Staubli VAL3: Rect3.dtx

public frame fReference = {x=1475.172, y=-187.34, z=-1030, rz=81.293, fatherId=world[0]}
public jointRx jPark = {j3=90, j5=90}
public jointRx jJoint = {j1=-21.01262, j2=66.00246, j3=79.8866, j5=34.11094, j6=162.86513}
public mdesc mNomSpeed = {blend=off}
public mdesc mSpeed[9]
  [0] = {tmax=75, rmax=100, leave=0.1, reach=0.1, blend=cartesian}
  [1] = {tmax=75, rmax=100, leave=0.1, reach=0.1, blend=cartesian}
  [2] = {tmax=75, rmax=100, leave=0.1, reach=0.1, blend=cartesian}
  [3] = {tmax=75, rmax=100, leave=0.1, reach=0.1, blend=cartesian}
  [4] = {tmax=75, rmax=100, leave=0.1, reach=0.1, blend=cartesian}
  [5] = {tmax=75, rmax=100, leave=0.1, reach=0.1, blend=cartesian}
  [6] = {tmax=75, rmax=100, leave=0.1, reach=0.1, blend=cartesian}
  [7] = {tmax=75, rmax=100, leave=0.1, reach=0.1, blend=cartesian}
  [8] = {tmax=75, rmax=100, leave=0.1, reach=0.1, blend=cartesian}
public num nTraj
num nTimeStop
num nTimeStart
num nMode
num nEtat
public pointRx pPoint[222]
  [0] = {x=-372, y=-44, z=100, rx=-180, rz=85.171, shoulder=lefty, elbow=epositive, wrist=wpositive, fatherId=fReference[0]}
  [1] = {x=-372, y=-44, rx=-180, rz=85.171, shoulder=lefty, elbow=epositive, wrist=wpositive, fatherId=fReference[0]}
  [2] = {x=-372, y=-44, rx=-180, rz=85.171, shoulder=lefty, elbow=epositive, wrist=wpositive, fatherId=fReference[0]}
  [3] = {x=-369.477, y=-73.864, rx=-180, rz=75.512, shoulder=lefty, elbow=epositive, wrist=wpositive, fatherId=fReference[0]}
  [4] = {x=-361.979, y=-102.881, rx=-180, rz=65.854, shoulder=lefty, elbow=epositive, wrist=wpositive, fatherId=fReference[0]}
  [5] = {x=-349.719, y=-130.229, rx=-180, rz=56.195, shoulder=lefty, elbow=epositive, wrist=wpositive, fatherId=fReference[0]}
  [6] = {x=-333.045, y=-155.133, rx=-180, rz=46.537, shoulder=lefty, elbow=epositive, wrist=wpositive, fatherId=fReference[0]}
  [7] = {x=-312.429, y=-176.886, rx=-180, rz=36.878, shoulder=lefty, elbow=epositive, wrist=wpositive, fatherId=fReference[0]}
  [8] = {x=-288.455, y=-194.872, rx=-180, rz=27.22, shoulder=lefty, elbow=epositive, wrist=wpositive, fatherId=fReference[0]}
  [9] = {x=-261.803, y=-208.58, rx=180, rz=17.561, shoulder=lefty, elbow=epositive, wrist=wpositive, fatherId=fReference[0]}
  [10] = {x=-233.23, y=-217.623, rx=-180, rz=7.903, shoulder=lefty, elbow=epositive, wrist=wpositive, fatherId=fReference[0]}
  [11] = {x=-203.544, y=-221.744, rx=180, rz=0.489, shoulder=lefty, elbow=epositive, wrist=wpositive, fatherId=fReference[0]}
  [12] = {x=-173.543, y=-222, rx=180, shoulder=lefty, elbow=epositive, wrist=wpositive, fatherId=fReference[0]}
  [13] = {x=-143.537, y=-222, rx=180, shoulder=lefty, elbow=epositive, wrist=wpositive, fatherId=fReference[0]}
  [14] = {x=-113.531, y=-222, rx=180, shoulder=lefty, elbow=epositive, wrist=wpositive, fatherId=fReference[0]}
  [15] = {x=-83.525, y=-222, rx=-180, shoulder=lefty, elbow=epositive, wrist=wpositive, fatherId=fReference[0]}
  [16] = {x=-53.519, y=-222, rx=180, shoulder=lefty, elbow=epositive, wrist=wpositive, fatherId=fReference[0]}
  [17] = {x=-23.513, y=-222, rx=180, shoulder=lefty, elbow=epositive, wrist=wpositive, fatherId=fReference[0]}
  [18] = {x=6.493, y=-222, rx=-180, shoulder=lefty, elbow=epositive, wrist=wpositive, fatherId=fReference[0]}
  [19] = {x=36.499, y=-222, rx=180, shoulder=lefty, elbow=epositive, wrist=wpositive, fatherId=fReference[0]}
  [20] = {x=66.504, y=-222, rx=180, shoulder=lefty, elbow=epositive, wrist=wpositive, fatherId=fReference[0]}
  [21] = {x=96.51, y=-222, rx=180, shoulder=lefty, elbow=epositive, wrist=wpositive, fatherId=fReference[0]}
  [22] = {x=126.516, y=-222, rx=180, shoulder=lefty, elbow=epositive, wrist=wpositive, fatherId=fReference[0]}
  [23] = {x=156.522, y=-222, rx=-180, shoulder=lefty, elbow=epositive, wrist=wpositive, fatherId=fReference[0]}
  [24] = {x=186.528, y=-222, rx=-180, rz=-2.723, shoulder=lefty, elbow=epositive, wrist=wpositive, fatherId=fReference[0]}
  [25] = {x=216.474, y=-220.576, rx=-180, rz=-12.083, shoulder=lefty, elbow=epositive, wrist=wpositive, fatherId=fReference[0]}
  [26] = {x=245.78, y=-214.302, rx=180, rz=-21.741, shoulder=lefty, elbow=epositive, wrist=wpositive, fatherId=fReference[0]}
  [27] = {x=273.619, y=-203.201, rx=-180, rz=-31.4, shoulder=lefty, elbow=epositive, wrist=wpositive, fatherId=fReference[0]}
  [28] = {x=299.2, y=-187.586, rx=180, rz=-41.058, shoulder=lefty, elbow=epositive, wrist=wpositive, fatherId=fReference[0]}
  [29] = {x=321.799, y=-167.901, rx=180, rz=-50.717, shoulder=lefty, elbow=epositive, wrist=wpositive, fatherId=fReference[0]}
  [30] = {x=340.775, y=-144.703, rx=180, rz=-60.375, shoulder=lefty, elbow=epositive, wrist=wpositive, fatherId=fReference[0]}
  [31] = {x=355.59, y=-118.65, rx=-180, rz=-70.034, shoulder=lefty, elbow=epositive, wrist=wpositive, fatherId=fReference[0]}
  [32] = {x=365.824, y=-90.481, rx=180, rz=-79.692, shoulder=lefty, elbow=epositive, wrist=wpositive, fatherId=fReference[0]}
  [33] = {x=371.187, y=-60.995, rx=180, rz=-88.446, shoulder=lefty, elbow=epositive, wrist=wpositive, fatherId=fReference[0]}
  [34] = {x=372, y=-31.015, rx=180, rz=-90, shoulder=lefty, elbow=epositive, wrist=wpositive, fatherId=fReference[0]}
  [35] = {x=372, y=-1.009, rx=180, rz=-90, shoulder=lefty, elbow=epositive, wrist=wpositive, fatherId=fReference[0]}
  [36] = {x=372, y=28.997, rx=-180, rz=-91.207, shoulder=lefty, elbow=epositive, wrist=wpositive, fatherId=fReference[0]}
  [37] = {x=371.368, y=58.985, rx=-180, rz=-99.658, shoulder=lefty, elbow=epositive, wrist=wpositive, fatherId=fReference[0]}
  [38] = {x=366.34, y=88.531, rx=-180, rz=-109.317, shoulder=lefty, elbow=epositive, wrist=wpositive, fatherId=fReference[0]}
  [39] = {x=356.426, y=116.814, rx=-180, rz=-118.975, shoulder=lefty, elbow=epositive, wrist=wpositive, fatherId=fReference[0]}
  [40] = {x=341.907, y=143.033, rx=-180, rz=-128.634, shoulder=lefty, elbow=epositive, wrist=wpositive, fatherId=fReference[0]}
  [41] = {x=323.195, y=166.444, rx=-180, rz=-138.292, shoulder=lefty, elbow=epositive, wrist=wpositive, fatherId=fReference[0]}
  [42] = {x=300.821, y=186.384, rx=180, rz=-147.951, shoulder=lefty, elbow=epositive, wrist=wpositive, fatherId=fReference[0]}
  [43] = {x=275.418, y=202.288, rx=180, rz=-157.609, shoulder=lefty, elbow=epositive, wrist=wpositive, fatherId=fReference[0]}
  [44] = {x=247.707, y=213.704, rx=-180, rz=-167.268, shoulder=lefty, elbow=epositive, wrist=wpositive, fatherId=fReference[0]}
  [45] = {x=218.474, y=220.309, rx=-180, rz=-176.767, shoulder=lefty, elbow=epositive, wrist=wpositive, fatherId=fReference[0]}
  [46] = {x=188.546, y=222, rx=-180, rz=180, shoulder=lefty, elbow=epositive, wrist=wpositive, fatherId=fReference[0]}
  [47] = {x=158.54, y=222, rx=-180, rz=180, shoulder=lefty, elbow=epositive, wrist=wpositive, fatherId=fReference[0]}
  [48] = {x=128.534, y=222, rx=180, rz=180, shoulder=lefty, elbow=epositive, wrist=wpositive, fatherId=fReference[0]}
  [49] = {x=98.528, y=222, rx=-180, rz=180, shoulder=lefty, elbow=epositive, wrist=wpositive, fatherId=fReference[0]}
  [50] = {x=68.522, y=222, rx=180, rz=180, shoulder=lefty, elbow=epositive, wrist=wpositive, fatherId=fReference[0]}
  [51] = {x=38.516, y=222, rx=-180, rz=180, shoulder=lefty, elbow=epositive, wrist=wpositive, fatherId=fReference[0]}
  [52] = {x=8.51, y=222, rx=-180, rz=180, shoulder=lefty, elbow=epositive, wrist=wpositive, fatherId=fReference[0]}
  [53] = {x=-21.496, y=222, rx=-180, rz=180, shoulder=lefty, elbow=epositive, wrist=wpositive, fatherId=fReference[0]}
  [54] = {x=-51.501, y=222, rx=-180, rz=180, shoulder=lefty, elbow=epositive, wrist=wpositive, fatherId=fReference[0]}
  [55] = {x=-81.507, y=222, rx=180, rz=180, shoulder=lefty, elbow=epositive, wrist=wpositive, fatherId=fReference[0]}
  [56] = {x=-111.513, y=222, rx=180, rz=-180, shoulder=lefty, elbow=epositive, wrist=wpositive, fatherId=fReference[0]}
  [57] = {x=-141.519, y=222, rx=180, rz=180, shoulder=lefty, elbow=epositive, wrist=wpositive, fatherId=fReference[0]}
  [58] = {x=-171.525, y=222, rx=-180, rz=179.696, shoulder=lefty, elbow=epositive, wrist=wpositive, fatherId=fReference[0]}
  [59] = {x=-201.529, y=221.841, rx=-180, rz=172.747, shoulder=lefty, elbow=epositive, wrist=wpositive, fatherId=fReference[0]}
  [60] = {x=-231.259, y=218.057, rx=-180, rz=163.088, shoulder=lefty, elbow=epositive, wrist=wpositive, fatherId=fReference[0]}
  [61] = {x=-259.934, y=209.338, rx=180, rz=153.43, shoulder=lefty, elbow=epositive, wrist=wpositive, fatherId=fReference[0]}
  [62] = {x=-286.739, y=195.933, rx=-180, rz=143.771, shoulder=lefty, elbow=epositive, wrist=wpositive, fatherId=fReference[0]}
  [63] = {x=-310.915, y=178.22, rx=180, rz=134.113, shoulder=lefty, elbow=epositive, wrist=wpositive, fatherId=fReference[0]}
  [64] = {x=-331.776, y=156.702, rx=180, rz=124.454, shoulder=lefty, elbow=epositive, wrist=wpositive, fatherId=fReference[0]}
  [65] = {x=-348.732, y=131.989, rx=180, rz=114.796, shoulder=lefty, elbow=epositive, wrist=wpositive, fatherId=fReference[0]}
  [66] = {x=-361.301, y=104.782, rx=180, rz=105.137, shoulder=lefty, elbow=epositive, wrist=wpositive, fatherId=fReference[0]}
  [67] = {x=-369.127, y=75.851, rx=180, rz=95.479, shoulder=lefty, elbow=epositive, wrist=wpositive, fatherId=fReference[0]}
  [68] = {x=-371.989, y=46.018, rx=180, rz=90.022, shoulder=lefty, elbow=epositive, wrist=wpositive, fatherId=fReference[0]}
  [69] = {x=-372, y=16.012, rx=-180, rz=90, shoulder=lefty, elbow=epositive, wrist=wpositive, fatherId=fReference[0]}
  [70] = {x=-372, y=-13.994, rx=-180, rz=90, shoulder=lefty, elbow=epositive, wrist=wpositive, fatherId=fReference[0]}
  [71] = {x=-372, y=-44, rx=-180, rz=90, shoulder=lefty, elbow=epositive, wrist=wpositive, fatherId=fReference[0]}
  [72] = {x=-372, y=-44, rx=-180, rz=90, shoulder=lefty, elbow=epositive, wrist=wpositive, fatherId=fReference[0]}
  [73] = {x=-372, y=-44, z=100, rx=-180, rz=90, shoulder=lefty, elbow=epositive, wrist=wpositive, fatherId=fReference[0]}
  [74] = {x=-372, y=-44, z=122, rx=-180, rz=90, shoulder=lefty, elbow=epositive, wrist=wpositive, fatherId=fReference[0]}
  [75] = {x=-372, y=-44, z=22, rx=-180, rz=90, shoulder=lefty, elbow=epositive, wrist=wpositive, fatherId=fReference[0]}
  [76] = {x=-372, y=-44, z=22, rx=-180, rz=90, shoulder=lefty, elbow=epositive, wrist=wpositive, fatherId=fReference[0]}
  [77] = {x=-372, y=-13.994, z=22, rx=-180, rz=90, shoulder=lefty, elbow=epositive, wrist=wpositive, fatherId=fReference[0]}
  [78] = {x=-372, y=16.012, z=22, rx=180, rz=90.022, shoulder=lefty, elbow=epositive, wrist=wpositive, fatherId=fReference[0]}
  [79] = {x=-371.989, y=46.018, z=22, rx=180, rz=95.479, shoulder=lefty, elbow=epositive, wrist=wpositive, fatherId=fReference[0]}
  [80] = {x=-369.127, y=75.851, z=22, rx=180, rz=105.137, shoulder=lefty, elbow=epositive, wrist=wpositive, fatherId=fReference[0]}
  [81] = {x=-361.301, y=104.782, z=22, rx=180, rz=114.796, shoulder=lefty, elbow=epositive, wrist=wpositive, fatherId=fReference[0]}
  [82] = {x=-348.732, y=131.989, z=22, rx=180, rz=124.454, shoulder=lefty, elbow=epositive, wrist=wpositive, fatherId=fReference[0]}
  [83] = {x=-331.776, y=156.702, z=22, rx=180, rz=134.113, shoulder=lefty, elbow=epositive, wrist=wpositive, fatherId=fReference[0]}
  [84] = {x=-310.915, y=178.22, z=22, rx=180, rz=143.771, shoulder=lefty, elbow=epositive, wrist=wpositive, fatherId=fReference[0]}
  [85] = {x=-286.739, y=195.933, z=22, rx=-180, rz=153.43, shoulder=lefty, elbow=epositive, wrist=wpositive, fatherId=fReference[0]}
  [86] = {x=-259.934, y=209.338, z=22, rx=-180, rz=163.088, shoulder=lefty, elbow=epositive, wrist=wpositive, fatherId=fReference[0]}
  [87] = {x=-231.259, y=218.057, z=22, rx=180, rz=172.747, shoulder=lefty, elbow=epositive, wrist=wpositive, fatherId=fReference[0]}
  [88] = {x=-201.529, y=221.841, z=22, rx=180, rz=179.696, shoulder=lefty, elbow=epositive, wrist=wpositive, fatherId=fReference[0]}
  [89] = {x=-171.525, y=222, z=22, rx=180, rz=180, shoulder=lefty, elbow=epositive, wrist=wpositive, fatherId=fReference[0]}
  [90] = {x=-141.519, y=222, z=22, rx=-180, rz=180, shoulder=lefty, elbow=epositive, wrist=wpositive, fatherId=fReference[0]}
  [91] = {x=-111.513, y=222, z=22, rx=180, rz=-180, shoulder=lefty, elbow=epositive, wrist=wpositive, fatherId=fReference[0]}
  [92] = {x=-81.507, y=222, z=22, rx=180, rz=180, shoulder=lefty, elbow=epositive, wrist=wpositive, fatherId=fReference[0]}
  [93] = {x=-51.501, y=222, z=22, rx=-180, rz=180, shoulder=lefty, elbow=epositive, wrist=wpositive, fatherId=fReference[0]}
  [94] = {x=-21.496, y=222, z=22, rx=-180, rz=180, shoulder=lefty, elbow=epositive, wrist=wpositive, fatherId=fReference[0]}
  [95] = {x=8.51, y=222, z=22, rx=-180, rz=180, shoulder=lefty, elbow=epositive, wrist=wpositive, fatherId=fReference[0]}
  [96] = {x=38.516, y=222, z=22, rx=180, rz=180, shoulder=lefty, elbow=epositive, wrist=wpositive, fatherId=fReference[0]}
  [97] = {x=68.522, y=222, z=22, rx=-180, rz=-180, shoulder=lefty, elbow=epositive, wrist=wpositive, fatherId=fReference[0]}
  [98] = {x=98.528, y=222, z=22, rx=-180, rz=180, shoulder=lefty, elbow=epositive, wrist=wpositive, fatherId=fReference[0]}
  [99] = {x=128.534, y=222, z=22, rx=-180, rz=180, shoulder=lefty, elbow=epositive, wrist=wpositive, fatherId=fReference[0]}
  [100] = {x=158.54, y=222, z=22, rx=-180, rz=180, shoulder=lefty, elbow=epositive, wrist=wpositive, fatherId=fReference[0]}
  [101] = {x=188.546, y=222, z=22, rx=-180, rz=-176.767, shoulder=lefty, elbow=epositive, wrist=wpositive, fatherId=fReference[0]}
  [102] = {x=218.474, y=220.309, z=22, rx=180, rz=-167.268, shoulder=lefty, elbow=epositive, wrist=wpositive, fatherId=fReference[0]}
  [103] = {x=247.707, y=213.704, z=22, rx=180, rz=-157.609, shoulder=lefty, elbow=epositive, wrist=wpositive, fatherId=fReference[0]}
  [104] = {x=275.418, y=202.288, z=22, rx=-180, rz=-147.951, shoulder=lefty, elbow=epositive, wrist=wpositive, fatherId=fReference[0]}
  [105] = {x=300.821, y=186.384, z=22, rx=-180, rz=-138.292, shoulder=lefty, elbow=epositive, wrist=wpositive, fatherId=fReference[0]}
  [106] = {x=323.195, y=166.444, z=22, rx=-180, rz=-128.634, shoulder=lefty, elbow=epositive, wrist=wpositive, fatherId=fReference[0]}
  [107] = {x=341.907, y=143.033, z=22, rx=-180, rz=-118.975, shoulder=lefty, elbow=epositive, wrist=wpositive, fatherId=fReference[0]}
  [108] = {x=356.426, y=116.814, z=22, rx=-180, rz=-109.317, shoulder=lefty, elbow=epositive, wrist=wpositive, fatherId=fReference[0]}
  [109] = {x=366.34, y=88.531, z=22, rx=-180, rz=-99.658, shoulder=lefty, elbow=epositive, wrist=wpositive, fatherId=fReference[0]}
  [110] = {x=371.368, y=58.985, z=22, rx=-180, rz=-91.207, shoulder=lefty, elbow=epositive, wrist=wpositive, fatherId=fReference[0]}
  [111] = {x=372, y=28.997, z=22, rx=180, rz=-90, shoulder=lefty, elbow=epositive, wrist=wpositive, fatherId=fReference[0]}
  [112] = {x=372, y=-1.009, z=22, rx=180, rz=-90, shoulder=lefty, elbow=epositive, wrist=wpositive, fatherId=fReference[0]}
  [113] = {x=372, y=-31.015, z=22, rx=180, rz=-88.446, shoulder=lefty, elbow=epositive, wrist=wpositive, fatherId=fReference[0]}
  [114] = {x=371.187, y=-60.995, z=22, rx=180, rz=-79.692, shoulder=lefty, elbow=epositive, wrist=wpositive, fatherId=fReference[0]}
  [115] = {x=365.824, y=-90.481, z=22, rx=180, rz=-70.034, shoulder=lefty, elbow=epositive, wrist=wpositive, fatherId=fReference[0]}
  [116] = {x=355.59, y=-118.65, z=22, rx=-180, rz=-60.375, shoulder=lefty, elbow=epositive, wrist=wpositive, fatherId=fReference[0]}
  [117] = {x=340.775, y=-144.703, z=22, rx=180, rz=-50.717, shoulder=lefty, elbow=epositive, wrist=wpositive, fatherId=fReference[0]}
  [118] = {x=321.799, y=-167.901, z=22, rx=180, rz=-41.058, shoulder=lefty, elbow=epositive, wrist=wpositive, fatherId=fReference[0]}
  [119] = {x=299.2, y=-187.586, z=22, rx=180, rz=-31.4, shoulder=lefty, elbow=epositive, wrist=wpositive, fatherId=fReference[0]}
  [120] = {x=273.619, y=-203.201, z=22, rx=180, rz=-21.741, shoulder=lefty, elbow=epositive, wrist=wpositive, fatherId=fReference[0]}
  [121] = {x=245.78, y=-214.302, z=22, rx=-180, rz=-12.083, shoulder=lefty, elbow=epositive, wrist=wpositive, fatherId=fReference[0]}
  [122] = {x=216.474, y=-220.576, z=22, rx=-180, rz=-2.723, shoulder=lefty, elbow=epositive, wrist=wpositive, fatherId=fReference[0]}
  [123] = {x=186.528, y=-222, z=22, rx=-180, shoulder=lefty, elbow=epositive, wrist=wpositive, fatherId=fReference[0]}
  [124] = {x=156.522, y=-222, z=22, rx=-180, shoulder=lefty, elbow=epositive, wrist=wpositive, fatherId=fReference[0]}
  [125] = {x=126.516, y=-222, z=22, rx=-180, shoulder=lefty, elbow=epositive, wrist=wpositive, fatherId=fReference[0]}
  [126] = {x=96.51, y=-222, z=22, rx=180, shoulder=lefty, elbow=epositive, wrist=wpositive, fatherId=fReference[0]}
  [127] = {x=66.504, y=-222, z=22, rx=180, shoulder=lefty, elbow=epositive, wrist=wpositive, fatherId=fReference[0]}
  [128] = {x=36.499, y=-222, z=22, rx=180, shoulder=lefty, elbow=epositive, wrist=wpositive, fatherId=fReference[0]}
  [129] = {x=6.493, y=-222, z=22, rx=-180, shoulder=lefty, elbow=epositive, wrist=wpositive, fatherId=fReference[0]}
  [130] = {x=-23.513, y=-222, z=22, rx=-180, shoulder=lefty, elbow=epositive, wrist=wpositive, fatherId=fReference[0]}
  [131] = {x=-53.519, y=-222, z=22, rx=180, shoulder=lefty, elbow=epositive, wrist=wpositive, fatherId=fReference[0]}
  [132] = {x=-83.525, y=-222, z=22, rx=-180, shoulder=lefty, elbow=epositive, wrist=wpositive, fatherId=fReference[0]}
  [133] = {x=-113.531, y=-222, z=22, rx=-180, shoulder=lefty, elbow=epositive, wrist=wpositive, fatherId=fReference[0]}
  [134] = {x=-143.537, y=-222, z=22, rx=180, shoulder=lefty, elbow=epositive, wrist=wpositive, fatherId=fReference[0]}
  [135] = {x=-173.543, y=-222, z=22, rx=180, rz=0.489, shoulder=lefty, elbow=epositive, wrist=wpositive, fatherId=fReference[0]}
  [136] = {x=-203.544, y=-221.744, z=22, rx=-180, rz=7.903, shoulder=lefty, elbow=epositive, wrist=wpositive, fatherId=fReference[0]}
  [137] = {x=-233.23, y=-217.623, z=22, rx=-180, rz=17.561, shoulder=lefty, elbow=epositive, wrist=wpositive, fatherId=fReference[0]}
  [138] = {x=-261.803, y=-208.58, z=22, rx=180, rz=27.22, shoulder=lefty, elbow=epositive, wrist=wpositive, fatherId=fReference[0]}
  [139] = {x=-288.455, y=-194.872, z=22, rx=-180, rz=36.878, shoulder=lefty, elbow=epositive, wrist=wpositive, fatherId=fReference[0]}
  [140] = {x=-312.429, y=-176.886, z=22, rx=180, rz=46.537, shoulder=lefty, elbow=epositive, wrist=wpositive, fatherId=fReference[0]}
  [141] = {x=-333.045, y=-155.133, z=22, rx=-180, rz=56.195, shoulder=lefty, elbow=epositive, wrist=wpositive, fatherId=fReference[0]}
  [142] = {x=-349.719, y=-130.229, z=22, rx=-180, rz=65.854, shoulder=lefty, elbow=epositive, wrist=wpositive, fatherId=fReference[0]}
  [143] = {x=-361.979, y=-102.881, z=22, rx=-180, rz=75.512, shoulder=lefty, elbow=epositive, wrist=wpositive, fatherId=fReference[0]}
  [144] = {x=-369.477, y=-73.864, z=22, rx=-180, rz=85.171, shoulder=lefty, elbow=epositive, wrist=wpositive, fatherId=fReference[0]}
  [145] = {x=-372, y=-44, z=22, rx=-180, rz=85.171, shoulder=lefty, elbow=epositive, wrist=wpositive, fatherId=fReference[0]}
  [146] = {x=-372, y=-44, z=22, rx=-180, rz=85.171, shoulder=lefty, elbow=epositive, wrist=wpositive, fatherId=fReference[0]}
  [147] = {x=-372, y=-44, z=122, rx=-180, rz=85.171, shoulder=lefty, elbow=epositive, wrist=wpositive, fatherId=fReference[0]}
  [148] = {x=-372, y=-44, z=144, rx=-180, rz=85.171, shoulder=lefty, elbow=epositive, wrist=wpositive, fatherId=fReference[0]}
  [149] = {x=-372, y=-44, z=44, rx=-180, rz=85.171, shoulder=lefty, elbow=epositive, wrist=wpositive, fatherId=fReference[0]}
  [150] = {x=-372, y=-44, z=44, rx=-180, rz=85.171, shoulder=lefty, elbow=epositive, wrist=wpositive, fatherId=fReference[0]}
  [151] = {x=-369.477, y=-73.864, z=44, rx=-180, rz=75.512, shoulder=lefty, elbow=epositive, wrist=wpositive, fatherId=fReference[0]}
  [152] = {x=-361.979, y=-102.881, z=44, rx=-180, rz=65.854, shoulder=lefty, elbow=epositive, wrist=wpositive, fatherId=fReference[0]}
  [153] = {x=-349.719, y=-130.229, z=44, rx=-180, rz=56.195, shoulder=lefty, elbow=epositive, wrist=wpositive, fatherId=fReference[0]}
  [154] = {x=-333.045, y=-155.133, z=44, rx=180, rz=46.537, shoulder=lefty, elbow=epositive, wrist=wpositive, fatherId=fReference[0]}
  [155] = {x=-312.429, y=-176.886, z=44, rx=-180, rz=36.878, shoulder=lefty, elbow=epositive, wrist=wpositive, fatherId=fReference[0]}
  [156] = {x=-288.455, y=-194.872, z=44, rx=180, rz=27.22, shoulder=lefty, elbow=epositive, wrist=wpositive, fatherId=fReference[0]}
  [157] = {x=-261.803, y=-208.58, z=44, rx=-180, rz=17.561, shoulder=lefty, elbow=epositive, wrist=wpositive, fatherId=fReference[0]}
  [158] = {x=-233.23, y=-217.623, z=44, rx=-180, rz=7.903, shoulder=lefty, elbow=epositive, wrist=wpositive, fatherId=fReference[0]}
  [159] = {x=-203.544, y=-221.744, z=44, rx=180, rz=0.489, shoulder=lefty, elbow=epositive, wrist=wpositive, fatherId=fReference[0]}
  [160] = {x=-173.543, y=-222, z=44, rx=180, shoulder=lefty, elbow=epositive, wrist=wpositive, fatherId=fReference[0]}
  [161] = {x=-143.537, y=-222, z=44, rx=-180, shoulder=lefty, elbow=epositive, wrist=wpositive, fatherId=fReference[0]}
  [162] = {x=-113.531, y=-222, z=44, rx=-180, shoulder=lefty, elbow=epositive, wrist=wpositive, fatherId=fReference[0]}
  [163] = {x=-83.525, y=-222, z=44, rx=-180, shoulder=lefty, elbow=epositive, wrist=wpositive, fatherId=fReference[0]}
  [164] = {x=-53.519, y=-222, z=44, rx=180, shoulder=lefty, elbow=epositive, wrist=wpositive, fatherId=fReference[0]}
  [165] = {x=-23.513, y=-222, z=44, rx=-180, shoulder=lefty, elbow=epositive, wrist=wpositive, fatherId=fReference[0]}
  [166] = {x=6.493, y=-222, z=44, rx=180, shoulder=lefty, elbow=epositive, wrist=wpositive, fatherId=fReference[0]}
  [167] = {x=36.499, y=-222, z=44, rx=-180, shoulder=lefty, elbow=epositive, wrist=wpositive, fatherId=fReference[0]}
  [168] = {x=66.504, y=-222, z=44, rx=180, shoulder=lefty, elbow=epositive, wrist=wpositive, fatherId=fReference[0]}
  [169] = {x=96.51, y=-222, z=44, rx=180, shoulder=lefty, elbow=epositive, wrist=wpositive, fatherId=fReference[0]}
  [170] = {x=126.516, y=-222, z=44, rx=180, shoulder=lefty, elbow=epositive, wrist=wpositive, fatherId=fReference[0]}
  [171] = {x=156.522, y=-222, z=44, rx=180, shoulder=lefty, elbow=epositive, wrist=wpositive, fatherId=fReference[0]}
  [172] = {x=186.528, y=-222, z=44, rx=180, rz=-2.723, shoulder=lefty, elbow=epositive, wrist=wpositive, fatherId=fReference[0]}
  [173] = {x=216.474, y=-220.576, z=44, rx=-180, rz=-12.083, shoulder=lefty, elbow=epositive, wrist=wpositive, fatherId=fReference[0]}
  [174] = {x=245.78, y=-214.302, z=44, rx=180, rz=-21.741, shoulder=lefty, elbow=epositive, wrist=wpositive, fatherId=fReference[0]}
  [175] = {x=273.619, y=-203.201, z=44, rx=180, rz=-31.4, shoulder=lefty, elbow=epositive, wrist=wpositive, fatherId=fReference[0]}
  [176] = {x=299.2, y=-187.586, z=44, rx=180, rz=-41.058, shoulder=lefty, elbow=epositive, wrist=wpositive, fatherId=fReference[0]}
  [177] = {x=321.799, y=-167.901, z=44, rx=-180, rz=-50.717, shoulder=lefty, elbow=epositive, wrist=wpositive, fatherId=fReference[0]}
  [178] = {x=340.775, y=-144.703, z=44, rx=180, rz=-60.375, shoulder=lefty, elbow=epositive, wrist=wpositive, fatherId=fReference[0]}
  [179] = {x=355.59, y=-118.65, z=44, rx=180, rz=-70.034, shoulder=lefty, elbow=epositive, wrist=wpositive, fatherId=fReference[0]}
  [180] = {x=365.824, y=-90.481, z=44, rx=180, rz=-79.692, shoulder=lefty, elbow=epositive, wrist=wpositive, fatherId=fReference[0]}
  [181] = {x=371.187, y=-60.995, z=44, rx=180, rz=-88.446, shoulder=lefty, elbow=epositive, wrist=wpositive, fatherId=fReference[0]}
  [182] = {x=372, y=-31.015, z=44, rx=180, rz=-90, shoulder=lefty, elbow=epositive, wrist=wpositive, fatherId=fReference[0]}
  [183] = {x=372, y=-1.009, z=44, rx=180, rz=-90, shoulder=lefty, elbow=epositive, wrist=wpositive, fatherId=fReference[0]}
  [184] = {x=372, y=28.997, z=44, rx=-180, rz=-91.207, shoulder=lefty, elbow=epositive, wrist=wpositive, fatherId=fReference[0]}
  [185] = {x=371.368, y=58.985, z=44, rx=-180, rz=-99.658, shoulder=lefty, elbow=epositive, wrist=wpositive, fatherId=fReference[0]}
  [186] = {x=366.34, y=88.531, z=44, rx=-180, rz=-109.317, shoulder=lefty, elbow=epositive, wrist=wpositive, fatherId=fReference[0]}
  [187] = {x=356.426, y=116.814, z=44, rx=-180, rz=-118.975, shoulder=lefty, elbow=epositive, wrist=wpositive, fatherId=fReference[0]}
  [188] = {x=341.907, y=143.033, z=44, rx=-180, rz=-128.634, shoulder=lefty, elbow=epositive, wrist=wpositive, fatherId=fReference[0]}
  [189] = {x=323.195, y=166.444, z=44, rx=-180, rz=-138.292, shoulder=lefty, elbow=epositive, wrist=wpositive, fatherId=fReference[0]}
  [190] = {x=300.821, y=186.384, z=44, rx=180, rz=-147.951, shoulder=lefty, elbow=epositive, wrist=wpositive, fatherId=fReference[0]}
  [191] = {x=275.418, y=202.288, z=44, rx=180, rz=-157.609, shoulder=lefty, elbow=epositive, wrist=wpositive, fatherId=fReference[0]}
  [192] = {x=247.707, y=213.704, z=44, rx=180, rz=-167.268, shoulder=lefty, elbow=epositive, wrist=wpositive, fatherId=fReference[0]}
  [193] = {x=218.474, y=220.309, z=44, rx=-180, rz=-176.767, shoulder=lefty, elbow=epositive, wrist=wpositive, fatherId=fReference[0]}
  [194] = {x=188.546, y=222, z=44, rx=-180, rz=180, shoulder=lefty, elbow=epositive, wrist=wpositive, fatherId=fReference[0]}
  [195] = {x=158.54, y=222, z=44, rx=-180, rz=-180, shoulder=lefty, elbow=epositive, wrist=wpositive, fatherId=fReference[0]}
  [196] = {x=128.534, y=222, z=44, rx=-180, rz=-180, shoulder=lefty, elbow=epositive, wrist=wpositive, fatherId=fReference[0]}
  [197] = {x=98.528, y=222, z=44, rx=-180, rz=180, shoulder=lefty, elbow=epositive, wrist=wpositive, fatherId=fReference[0]}
  [198] = {x=68.522, y=222, z=44, rx=180, rz=-180, shoulder=lefty, elbow=epositive, wrist=wpositive, fatherId=fReference[0]}
  [199] = {x=38.516, y=222, z=44, rx=-180, rz=180, shoulder=lefty, elbow=epositive, wrist=wpositive, fatherId=fReference[0]}
  [200] = {x=8.51, y=222, z=44, rx=180, rz=-180, shoulder=lefty, elbow=epositive, wrist=wpositive, fatherId=fReference[0]}
  [201] = {x=-21.496, y=222, z=44, rx=-180, rz=180, shoulder=lefty, elbow=epositive, wrist=wpositive, fatherId=fReference[0]}
  [202] = {x=-51.501, y=222, z=44, rx=-180, rz=180, shoulder=lefty, elbow=epositive, wrist=wpositive, fatherId=fReference[0]}
  [203] = {x=-81.507, y=222, z=44, rx=-180, rz=180, shoulder=lefty, elbow=epositive, wrist=wpositive, fatherId=fReference[0]}
  [204] = {x=-111.513, y=222, z=44, rx=180, rz=-180, shoulder=lefty, elbow=epositive, wrist=wpositive, fatherId=fReference[0]}
  [205] = {x=-141.519, y=222, z=44, rx=180, rz=180, shoulder=lefty, elbow=epositive, wrist=wpositive, fatherId=fReference[0]}
  [206] = {x=-171.525, y=222, z=44, rx=-180, rz=179.696, shoulder=lefty, elbow=epositive, wrist=wpositive, fatherId=fReference[0]}
  [207] = {x=-201.529, y=221.841, z=44, rx=180, rz=172.747, shoulder=lefty, elbow=epositive, wrist=wpositive, fatherId=fReference[0]}
  [208] = {x=-231.259, y=218.057, z=44, rx=180, rz=163.088, shoulder=lefty, elbow=epositive, wrist=wpositive, fatherId=fReference[0]}
  [209] = {x=-259.934, y=209.338, z=44, rx=180, rz=153.43, shoulder=lefty, elbow=epositive, wrist=wpositive, fatherId=fReference[0]}
  [210] = {x=-286.739, y=195.933, z=44, rx=180, rz=143.771, shoulder=lefty, elbow=epositive, wrist=wpositive, fatherId=fReference[0]}
  [211] = {x=-310.915, y=178.22, z=44, rx=180, rz=134.113, shoulder=lefty, elbow=epositive, wrist=wpositive, fatherId=fReference[0]}
  [212] = {x=-331.776, y=156.702, z=44, rx=180, rz=124.454, shoulder=lefty, elbow=epositive, wrist=wpositive, fatherId=fReference[0]}
  [213] = {x=-348.732, y=131.989, z=44, rx=180, rz=114.796, shoulder=lefty, elbow=epositive, wrist=wpositive, fatherId=fReference[0]}
  [214] = {x=-361.301, y=104.782, z=44, rx=180, rz=105.137, shoulder=lefty, elbow=epositive, wrist=wpositive, fatherId=fReference[0]}
  [215] = {x=-369.127, y=75.851, z=44, rx=180, rz=95.479, shoulder=lefty, elbow=epositive, wrist=wpositive, fatherId=fReference[0]}
  [216] = {x=-371.989, y=46.018, z=44, rx=180, rz=90.022, shoulder=lefty, elbow=epositive, wrist=wpositive, fatherId=fReference[0]}
  [217] = {x=-372, y=16.012, z=44, rx=-180, rz=90, shoulder=lefty, elbow=epositive, wrist=wpositive, fatherId=fReference[0]}
  [218] = {x=-372, y=-13.994, z=44, rx=-180, rz=90, shoulder=lefty, elbow=epositive, wrist=wpositive, fatherId=fReference[0]}
  [219] = {x=-372, y=-44, z=44, rx=-180, rz=90, shoulder=lefty, elbow=epositive, wrist=wpositive, fatherId=fReference[0]}
  [220] = {x=-372, y=-44, z=44, rx=-180, rz=90, shoulder=lefty, elbow=epositive, wrist=wpositive, fatherId=fReference[0]}
  [221] = {x=-372, y=-44, z=144, rx=-180, rz=90, shoulder=lefty, elbow=epositive, wrist=wpositive, fatherId=fReference[0]}
public tool tTool = {z=470, fatherId=flange[0], ioLink=valve1}
aio Tpompe = {link=CanIO\RemIO\remio0_QW}
dio doPompe = {link=CanIO\RemIO\remio0_Q}
dio doValve1 = {link=valve1}
dio doValve2 = {link=valve2}
num nTension = 3
num nTObtOpen = 6
num nTPompeOff
num nTPompeOn = 2
